{attribute addProperty BoxType "EP6002-0002-0017"}
{attribute addProperty Id "COM_TxPDO_Map_Inputs_ChannelAT %I*ARRAY[0..1] OF COM_TxPDO_Map_Inputs_Channel_4EE430B6384480COM_RxPDO_Map_Outputs_ChannelAT %Q*ARRAY[0..1] OF COM_RxPDO_Map_Outputs_Channel_CEA6CFDD384480WcStateAT %I*WcState_F855686C1620InfoDataAT %I*InfoData_BC63D37F80100"}
{attribute addProperty CRC "4210475582"}
{attribute addProperty SizeInBites "864"}
{attribute addProperty SizeInBytes "108"}
TYPE EP6002_6961C256 :
STRUCT
	{attribute addProperty Name "COM_TxPDO_Map_Inputs_Channel"}
	COM_TxPDO_Map_Inputs_Channel : ARRAY[0..1] OF COM_TxPDO_Map_Inputs_Channel_4EE430B6;
	{attribute addProperty Name "COM_RxPDO_Map_Outputs_Channel"}
	COM_RxPDO_Map_Outputs_Channel : ARRAY[0..1] OF COM_RxPDO_Map_Outputs_Channel_CEA6CFDD;
	{attribute addProperty Name "WcState"}
	WcState : WcState_F855686C;
	{attribute addProperty Name "InfoData"}
	InfoData : InfoData_BC63D37F;
END_STRUCT
END_TYPE

(* stored: Version 1.2.0.0, ProductVersion 3.1.4024.9
   DUT EP6002_6961C256: Id {2aca978d-cf64-420b-a700-8a2fd317e2e1} *)
